FUNCTION_BLOCK MY_X2Y2_J (* Compute X^2-Y^2 in ST *)
  (* Standard: 61499-1 *)
  (* Version 0.0, 2002-09-24, JHC, Rockwell Automation, Derived from FB_X2Y2_J. *)
  (* Compiler header: package fb.rt.student; *)
  (* Compiler Java IBM Jikes 1.0.6 *)
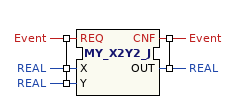
  EVENT_INPUT
    REQ WITH X, Y;
  END_EVENT
  EVENT_OUTPUT
    CNF WITH OUT;
  END_EVENT
  VAR_INPUT
    X : REAL;
    Y : REAL;
  END_VAR
  VAR_OUTPUT
    OUT : REAL;
  END_VAR
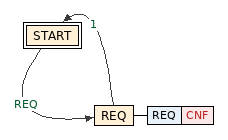
  EC_STATES
    START;
    REQ : REQ -> CNF;
  END_STATES
  EC_TRANSITIONS
    START TO REQ := REQ;
    REQ TO START := 1;
  END_TRANSITIONS
  ALGORITHM REQ IN Java:
OUT.value=(float)((X.value*X.value)+(Y.value*Y.value));
  END_ALGORITHM
END_FUNCTION_BLOCK
